(* PLC project Unnamed, Unknown Unnamed 1 *)
(* stored: creationDateTime 2013-01-29T14:01:00, modificationDateTime 2017-06-08T15:59:13 *)

FUNCTION WORDS_TO_REAL : REAL
  VAR_INPUT
    WORD_1 : WORD;
    WORD_2 : WORD;
  END_VAR

                        
                     {{
                     #include <stdint.h>
                     typedef uint32_t u32;
                     typedef uint16_t u16;
                     typedef uint8_t u8;
                     u32 out_value = WORD_1 | (WORD_2 << 16);
                     WORDS_TO_REAL = *(float*)&out_value;
                     }}
                    
                    
END_FUNCTION
